(* IEC 61131-3 sources: teller/JD_Teller_LC2_V11/Class/Count_To, 1 file *)

(* ---- Count_To.st ---- *)
(*!
<Class
	Name               = "Count_To"
	Revision           = "0.0"
	RealtimeTask       = "false"
	CyclicTask         = "false"
	BackgroundTask     = "true"
	DefBackground      = "100 ms"
	Sigmatek           = "false"
	OSInterface        = "false"
	HighPriority       = "false"
	Automatic          = "false"
	UpdateMode         = "Prescan"
	SharedCommandTable = "true"
	Objectsize         = "(284,120)">
	<Channels>
		<Server Name="ClassSvr" Visualized="false" Initialize="false" WriteProtected="true" Retentive="false"/>
		<Server Name="Count_To_3" Visualized="true" Initialize="false" WriteProtected="false" Retentive="false"/>
		<Server Name="Count_To_5" Visualized="true" Initialize="false" WriteProtected="false" Retentive="false"/>
	</Channels>
</Class>
*)
Count_To : CLASS
  //Servers:
	ClassSvr 	: SvrChCmd_DINT;
	Count_To_3 	: SvrCh_DINT;
	Count_To_5 	: SvrCh_DINT;
  //Clients:
  //Variables:
  //Functions:

	FUNCTION VIRTUAL GLOBAL Background
		VAR_INPUT
			EAX 	: UDINT;
		END_VAR
		VAR_OUTPUT
			state (EAX) 	: UDINT;
		END_VAR;
  //Tables:
	FUNCTION @STD
		VAR_OUTPUT
			ret_code	: CONFSTATES;
		END_VAR;
	FUNCTION GLOBAL TAB @CT_;
END_CLASS;

FUNCTION VIRTUAL GLOBAL Count_To::Background
	VAR_INPUT
		EAX 	: UDINT;
	END_VAR
	VAR_OUTPUT
		state (EAX) 	: UDINT;
	END_VAR

// Twee tellers die tot 3 en 5 tellen om geanimeerde plaatjes te maken in LSE

  Count_To_3 +=1;
  Count_To_5 +=1;

if Count_To_3 >3 then
  Count_To_3 :=1;
end_if;

if Count_To_5 >5 then
  Count_To_5 :=1;
end_if;

	state := READY;

END_FUNCTION
